// TIA Portal V20 export
FUNCTION "LER_TransferAndGenerate" : Void   // FC78, LAD
// stored: Access Published, SetENOAutomatically false
   VAR_INPUT
      partDataA : "LER_typePartData";
      transferCondition : Bool;
      partDetect : Bool;
      generateEmNumber : Int;
   END_VAR
   VAR_OUTPUT
      partDataB : "LER_typePartData";
      DataDelete : Bool;
   END_VAR
   VAR_TEMP
      tempRetVal : Int;
   END_VAR
BEGIN

REGION Network 1: Data Transfer
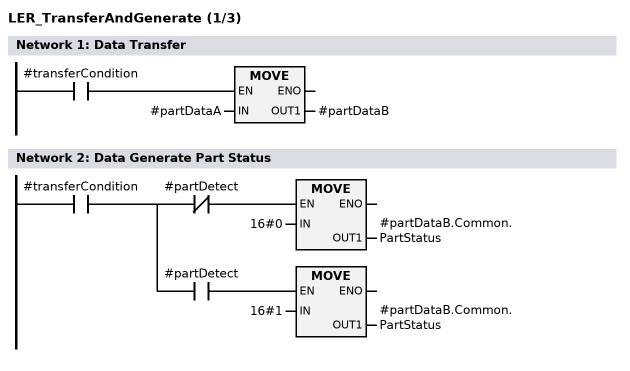
   RUNG wire#powerrail
      Contact( #transferCondition )
      Move(in := #partDataA, out1 => #partDataB)
   END_RUNG
   // the same network as SCL:
   IF #transferCondition THEN #partDataB := #partDataA; END_IF;
END_REGION

REGION Network 2: Data Generate Part Status
   RUNG wire#powerrail
      Contact( #transferCondition )
      wire#w1
      I_Contact( #partDetect )
      Move(in := 16#0, out1 => #partDataB.Common.PartStatus)
   END_RUNG
   RUNG wire#w1
      Contact( #partDetect )
      Move(in := 16#1, out1 => #partDataB.Common.PartStatus)
   END_RUNG
   // the same network as SCL:
   IF #transferCondition AND NOT #partDetect THEN #partDataB.Common.PartStatus := 16#0; END_IF;
   IF #transferCondition AND #partDetect THEN #partDataB.Common.PartStatus := 16#1; END_IF;
END_REGION

REGION Network 3: Data Generate Last Machine Number
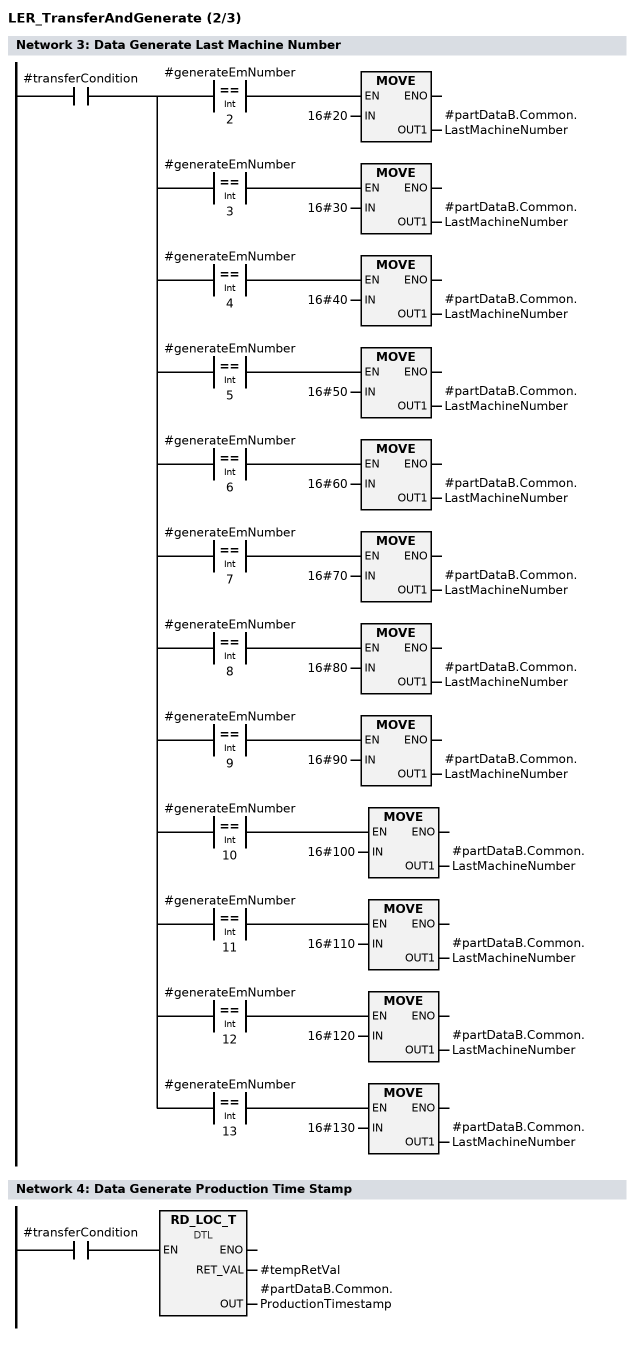
   RUNG wire#powerrail
      Contact( #transferCondition )
      wire#w1
      { S7_Templates := "SrcType := Int" } EQ_Contact(in1 := #generateEmNumber, in2 := 2)
      Move(in := 16#20, out1 => #partDataB.Common.LastMachineNumber)
   END_RUNG
   RUNG wire#w1
      { S7_Templates := "SrcType := Int" } EQ_Contact(in1 := #generateEmNumber, in2 := 3)
      Move(in := 16#30, out1 => #partDataB.Common.LastMachineNumber)
   END_RUNG
   RUNG wire#w1
      { S7_Templates := "SrcType := Int" } EQ_Contact(in1 := #generateEmNumber, in2 := 4)
      Move(in := 16#40, out1 => #partDataB.Common.LastMachineNumber)
   END_RUNG
   RUNG wire#w1
      { S7_Templates := "SrcType := Int" } EQ_Contact(in1 := #generateEmNumber, in2 := 5)
      Move(in := 16#50, out1 => #partDataB.Common.LastMachineNumber)
   END_RUNG
   RUNG wire#w1
      { S7_Templates := "SrcType := Int" } EQ_Contact(in1 := #generateEmNumber, in2 := 6)
      Move(in := 16#60, out1 => #partDataB.Common.LastMachineNumber)
   END_RUNG
   RUNG wire#w1
      { S7_Templates := "SrcType := Int" } EQ_Contact(in1 := #generateEmNumber, in2 := 7)
      Move(in := 16#70, out1 => #partDataB.Common.LastMachineNumber)
   END_RUNG
   RUNG wire#w1
      { S7_Templates := "SrcType := Int" } EQ_Contact(in1 := #generateEmNumber, in2 := 8)
      Move(in := 16#80, out1 => #partDataB.Common.LastMachineNumber)
   END_RUNG
   RUNG wire#w1
      { S7_Templates := "SrcType := Int" } EQ_Contact(in1 := #generateEmNumber, in2 := 9)
      Move(in := 16#90, out1 => #partDataB.Common.LastMachineNumber)
   END_RUNG
   RUNG wire#w1
      { S7_Templates := "SrcType := Int" } EQ_Contact(in1 := #generateEmNumber, in2 := 10)
      Move(in := 16#100, out1 => #partDataB.Common.LastMachineNumber)
   END_RUNG
   RUNG wire#w1
      { S7_Templates := "SrcType := Int" } EQ_Contact(in1 := #generateEmNumber, in2 := 11)
      Move(in := 16#110, out1 => #partDataB.Common.LastMachineNumber)
   END_RUNG
   RUNG wire#w1
      { S7_Templates := "SrcType := Int" } EQ_Contact(in1 := #generateEmNumber, in2 := 12)
      Move(in := 16#120, out1 => #partDataB.Common.LastMachineNumber)
   END_RUNG
   RUNG wire#w1
      { S7_Templates := "SrcType := Int" } EQ_Contact(in1 := #generateEmNumber, in2 := 13)
      Move(in := 16#130, out1 => #partDataB.Common.LastMachineNumber)
   END_RUNG
   // the same network as SCL:
   IF #transferCondition AND (#generateEmNumber = 2) THEN
       #partDataB.Common.LastMachineNumber := 16#20;
   END_IF;
   IF #transferCondition AND (#generateEmNumber = 3) THEN
       #partDataB.Common.LastMachineNumber := 16#30;
   END_IF;
   IF #transferCondition AND (#generateEmNumber = 4) THEN
       #partDataB.Common.LastMachineNumber := 16#40;
   END_IF;
   IF #transferCondition AND (#generateEmNumber = 5) THEN
       #partDataB.Common.LastMachineNumber := 16#50;
   END_IF;
   IF #transferCondition AND (#generateEmNumber = 6) THEN
       #partDataB.Common.LastMachineNumber := 16#60;
   END_IF;
   IF #transferCondition AND (#generateEmNumber = 7) THEN
       #partDataB.Common.LastMachineNumber := 16#70;
   END_IF;
   IF #transferCondition AND (#generateEmNumber = 8) THEN
       #partDataB.Common.LastMachineNumber := 16#80;
   END_IF;
   IF #transferCondition AND (#generateEmNumber = 9) THEN
       #partDataB.Common.LastMachineNumber := 16#90;
   END_IF;
   IF #transferCondition AND (#generateEmNumber = 10) THEN
       #partDataB.Common.LastMachineNumber := 16#100;
   END_IF;
   IF #transferCondition AND (#generateEmNumber = 11) THEN
       #partDataB.Common.LastMachineNumber := 16#110;
   END_IF;
   IF #transferCondition AND (#generateEmNumber = 12) THEN
       #partDataB.Common.LastMachineNumber := 16#120;
   END_IF;
   IF #transferCondition AND (#generateEmNumber = 13) THEN
       #partDataB.Common.LastMachineNumber := 16#130;
   END_IF;
END_REGION

REGION Network 4: Data Generate Production Time Stamp
   RUNG wire#powerrail
      Contact( #transferCondition )
      { S7_Templates := "date_type := DTL" } RD_LOC_T(RET_VAL => #tempRetVal, OUT => #partDataB.Common.ProductionTimestamp)
   END_RUNG
   // the same network as SCL:
   IF #transferCondition THEN #tempRetVal := RD_LOC_T(OUT => #partDataB.Common.ProductionTimestamp); END_IF;
END_REGION

REGION Network 5: Deleting Data
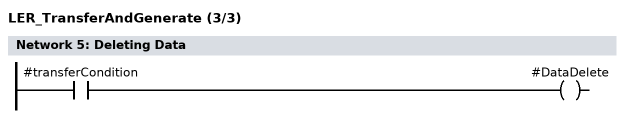
   RUNG wire#powerrail
      Contact( #transferCondition )
      Coil( #DataDelete )
   END_RUNG
   // the same network as SCL:
   #DataDelete := #transferCondition;
END_REGION
END_FUNCTION
